FUNCTION_BLOCK FB_CamIn_empty
VAR_INPUT
  Master            : REFERENCE TO Tc2_MC2.AXIS_REF;
  Slave             : REFERENCE TO Tc2_MC2.AXIS_REF; 
  Execute           : BOOL;
  MasterOffset      : REAL; 
  SlaveOffset       : REAL; 
  MasterScaling     : REAL;
  SlaveScaling      : REAL;
  StartMode         : INT;
  CamTableID        : UDINT;
END_VAR
VAR_OUTPUT
  Busy              : BOOL;
  Error             : BOOL;
  Done              : BOOL;
  InSync            : BOOL;
  ErrorId           : UDINT;
END_VAR
VAR
END_VAR


Error   := TRUE;
ErrorId := 9999; // function is not activated by compiler def CAM

END_FUNCTION_BLOCK

(* stored: Version 1.1.0.1, ProductVersion 3.1.4024.9
   POU FB_CamIn_empty: Id {41c3a096-0f5f-0263-3b7e-37393841b3af}, SpecialFunc None *)
